TYPE ST_TsGroupInfo :
STRUCT

	nState	 	 							:USINT;
	nDiag 	 								:USINT;

END_STRUCT
END_TYPE
(* End *)

(* stored: Version 1.1.0.1, ProductVersion 3.1.4022.16
   DUT ST_TsGroupInfo: Id {70377ce2-5274-424e-ad50-b6ada875c2fc} *)
